FUNCTION_BLOCK FB_TOR_Standard EXTENDS FB_TOR_Base
//////////////////
//  Circuit Breaker
//////////////////

VAR_INPUT PERSISTENT
	// Parameters of the Object (instance/model specific) 
		
		
END_VAR

VAR_OUTPUT
	//Child objects
	
END_VAR

VAR_INPUT
	// I/O Inputs 		                                     				
		
END_VAR

VAR
	//M_ALARMMANAGEMENT VARIABLES//
		
MesDataExd			: TOR_Standard ;  

	
END_VAR

METHOD M_AlarmManagement
//////////////////
// Manages Door sensor alarms and warnings
/////////////////

VAR 
	// Method local variables (reinitialized at each cycle) 
	FB_AlarmCodeManager : FB_AlarmCodeManager ; 


END_VAR

// ALARM CODE //
	FB_AlarmCodeManager(
 		bAlarm1			:= FALSE,    					// 
		bAlarm2			:= FALSE, 						// 
		bAlarm3			:= FALSE, 						// 
		bAlarm4			:= FALSE, 						// 
		bAlarm5			:= FALSE,       				//
		bAlarm6			:= FALSE,       				//
		bAlarm7			:= FALSE,       				//
		bAlarm8			:= FALSE,       				//
		bAlarm9			:= FALSE,       				//
		bAlarm10		:= FALSE,       				//
		bAlarm11		:= FALSE,       				//
		bAlarm12		:= FALSE,         				//
		bAlarm13		:= FALSE,         				//
		bAlarm14		:= FALSE,         				//
		bAlarm15		:= FALSE,         				//
		wAlarmCode		=>MesDataExd.MesData.MesAlarmCode);

// WARNING CODE //
	FB_AlarmCodeManager(
		bAlarm1			:= FALSE,    			// 
		bAlarm2			:= FALSE, 				//  
		bAlarm3			:= FALSE, 				//  
		bAlarm4			:= FALSE, 				//  
		bAlarm5			:= FALSE,               //
		bAlarm6			:= FALSE,               //
		bAlarm7			:= FALSE,               //
		bAlarm8			:= FALSE,               //
		bAlarm9			:= FALSE,               //
		bAlarm10		:= FALSE,               //
		bAlarm11		:= FALSE,               //
		bAlarm12		:= FALSE,               //
		bAlarm13		:= FALSE,               //
		bAlarm14		:= FALSE,               //
		bAlarm15		:= FALSE,               //
		wAlarmCode		=>MesDataExd.MesData.MesWarningCode);

// EVENT CODE //
	FB_AlarmCodeManager(
		bAlarm1			:= MesDataExd.MesData.MesAlarmState, 			//  CB is opened
		bAlarm2			:= FALSE, 							// 
		bAlarm3			:= FALSE, 							//  
		bAlarm4			:= FALSE, 							// 
		bAlarm5			:= FALSE,                           //
		bAlarm6			:= FALSE,                           //
		bAlarm7			:= FALSE,                           //
		bAlarm8			:= FALSE,                           //
		bAlarm9			:= FALSE,                           //
		bAlarm10		:= FALSE,                           //
		bAlarm11		:= FALSE,                           //
		bAlarm12		:= FALSE,                           //
		bAlarm13		:= FALSE,                           //
		bAlarm14		:= FALSE,                           //
		bAlarm15		:= FALSE,                           //
		wAlarmCode		=>MesDataExd.MesData.MesEventCode);
END_METHOD

METHOD M_StateManager
//////////////////
// Detect when fire occurs
/////////////////

VAR 
	// Method local variables (reinitialized at each cycle)
 	MesStateInterm1 : BOOL;
	MesStateInterm2 : BOOL;
END_VAR

IF ParamCableCutSecurity THEN
	MesStateInterm1 := NOT IN_MesState1_IO ; 
	MesStateInterm2 := NOT IN_MesState2_IO ; 
ELSE 
	MesStateInterm1 := IN_MesState1_IO;
	MesStateInterm2 := IN_MesState2_IO;
END_IF

IF ParamNbSensors = 1 THEN 
	MesStateInterm2 := MesStateInterm1 ;
END_IF

IF ParamAtleastOne THEN 
MesDataExd.MesData.MesAlarmState := MesStateInterm1 OR MesStateInterm2 ; 
ELSE
MesDataExd.MesData.MesAlarmState := MesStateInterm1 AND MesStateInterm2 ; 
END_IF

R_TRIGAlarm(CLK:= MesDataExd.MesData.MesAlarmState ) ; 
IF R_TRIGAlarm.Q THEN
	MesCountAlarm :=  MIN(MesCountAlarm + 1 ,4294967295 ) ; 
ELSIF IN_ResetCounter THEN 
	MesCountAlarm := 0 ; 
END_IF

MesDataExd.MesData.MesCountAlarm	:= MesCountAlarm ;
END_METHOD

END_FUNCTION_BLOCK

(* stored: Version 1.1.0.1, ProductVersion 3.1.4024.6
   POU FB_TOR_Standard: Id {bd19afec-f9b6-454b-80ac-d9303ba60605}, SpecialFunc None
   Method M_AlarmManagement: Id {a2ebc626-6800-42a4-8b43-8672f1c366d1}
   Method M_StateManager: Id {6c87c2a1-79d7-44e0-be60-f7d08976cf7c} *)
